// Mitsubishi GX Works2 project: 세탁기+탈수기   PLC: Q03UDV

PROGRAM MAIN
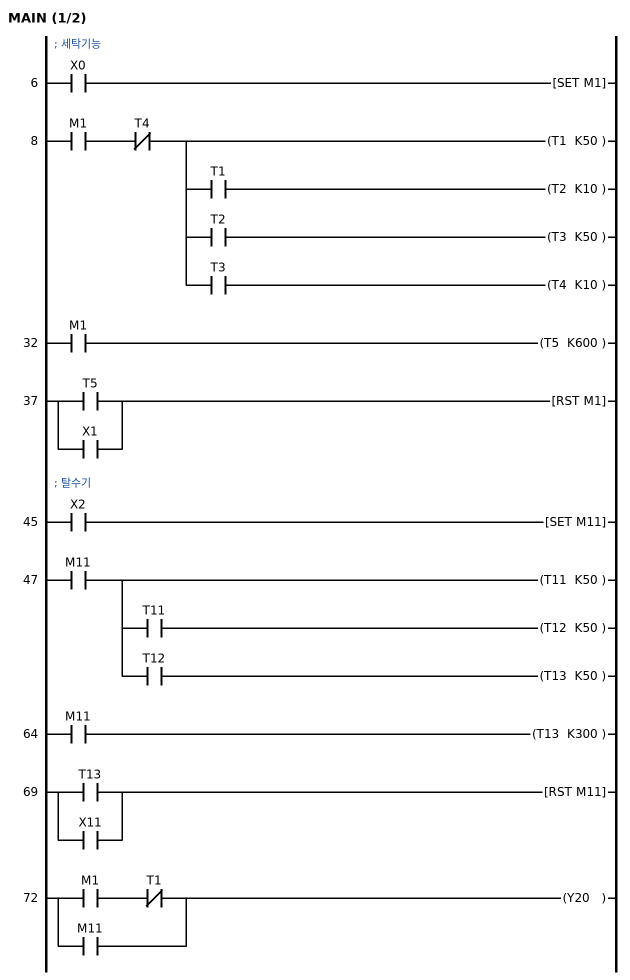
; 세탁기능
6     LD      X0
      SET     M1
8     LD      M1
      ANI     T4
      OUT     T1 K50
      MPS
      AND     T1
      OUT     T2 K10
      MRD
      AND     T2
      OUT     T3 K50
      MPP
      AND     T3
      OUT     T4 K10
32    LD      M1
      OUT     T5 K600
37    LD      T5
      OR      X1
      RST     M1
; 탈수기
45    LD      X2
      SET     M11
47    LD      M11
      OUT     T11 K50
      MPS
      AND     T11
      OUT     T12 K50
      MPP
      AND     T12
      OUT     T13 K50
64    LD      M11
      OUT     T13 K300
69    LD      T13
      OR      X11
      RST     M11
72    LD      M1
      ANI     T1
      OR      M11
      OUT     Y20
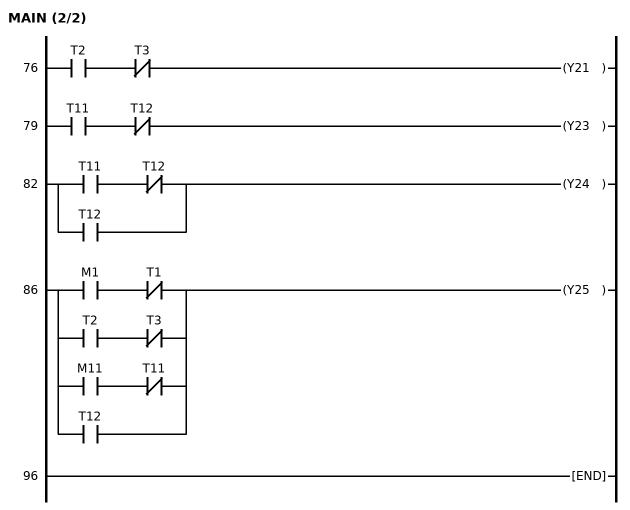
76    LD      T2
      ANI     T3
      OUT     Y21
79    LD      T11
      ANI     T12
      OUT     Y23
82    LD      T11
      ANI     T12
      OR      T12
      OUT     Y24
86    LD      M1
      ANI     T1
      LD      T2
      ANI     T3
      ORB
      LD      M11
      ANI     T11
      ORB
      OR      T12
      OUT     Y25
96    END
END_PROGRAM
